FUNCTION FC10 : VOID
//QAVGN

VAR_TEMP
    Temp:REAL;
END_VAR

VAR_INPUT
    IN1:REAL;
    IN2:REAL;
END_VAR

VAR_OUTPUT
    OUT:REAL;
END_VAR
    Temp:=IN1+IN2;
    OUT:=Temp/2;
END_FUNCTION

